{attribute 'GeneratedUsingTerminal: EK1122-0000-0018'}
{attribute addProperty BoxType "EK1122-0000-0018"}
{attribute addProperty Id "R4_FESTO_CMMP_AS_V4p0_CiA402CMMP_93B92D5237RH_EK1100RH_EK1100_A5940DFE232"}
{attribute addProperty CRC "625235105"}
{attribute addProperty Size "269"}
{attribute addProperty Name "R4_A2_EC (EK1122)"}
TYPE R4_A2_EC_EK1122_254454A1 EXTENDS EK1122_1FC0878B :
STRUCT
    {attribute addProperty Name "R4_FESTO (CMMP-AS V4p0 CiA402)"}
    {attribute addProperty PreviousPort "R4_A2_EC (EK1122) : D"}
    {attribute addProperty SyncUnit "default"}
    R4_FESTO_CMMP_AS_V4p0_CiA402 : CMMP_93B92D52;
    {attribute addProperty Name "RH (EK1100)"}
    {attribute addProperty PreviousPort "R4_A2_EC (EK1122) : B"}
    {attribute addProperty SyncUnit "default"}
    RH_EK1100 : RH_EK1100_A5940DFE;
END_STRUCT
END_TYPE

(* stored: Version 1.2.0.0, ProductVersion 3.1.4024.11
   DUT R4_A2_EC_EK1122_254454A1: Id {79b5ba1b-605d-0073-19f2-9c72de1d35dd} *)
